(* Logix 5000 project; controller DispersionPlc vendor 1 type 14 code 108 rev 34.11; software revision 34.01; part 14 of 22 *)
(* tags used below, declared in another part *)
   _JISdebug : DINT;
   AFI : BOOL;
   Circulation_Timer_Continue : BOOL;
   Estop_Disp : ALIAS FOR Local:3:I.Data.1;
   FC_4302_1 : AStd_PIDInterface;
   FC_4302_1_AOI : AStd_PIDInterface_AOI;
   FC_4302_1_PID : PID_ENHANCED;
   FC_4305_xx : AStd_PIDInterface;
   FC_4305_xx_AOI : AStd_PIDInterface_AOI;
   FC_4305_xx_PID : PID_ENHANCED;
   FCV_4302_1 : AStd_VlvModulating;
   FIT_4302_2 : AStd_AnalogInput;
   FIT_4305_xx : AStd_AnalogInput;
   FQIC_4302_11_Calc_TransferSetpoint : DINT;
   FQIC_4302_11_CurrentTrasferredLb : DINT;
   FQIC_4302_11_Pulse : BOOL;
   FQIC_4302_11_PulseCounter : COUNTER;
   FQIC_4302_11_PulseToLbFactor : DINT;
   FQIC_4302_11_Reset : BOOL;
   FQIC_4302_11_TransferOffset : DINT;
   FQIC_4302_11_TransferSetpoint : DINT;
   FQIC_4302_11_TransferStopValueLb : DINT;
   FV_4305_xx : AStd_VlvModulating;
   GenPurp : AStd_GeneralPurp;
   LS_4302_High : BOOL;
   One_Shots : DINT;
   P_4305 : AStd_FVNR;
   P_S52_2_OpenC : ALIAS FOR Local:1:O.Data[12].14;
   PLCStatus : AStd_PLCStatus;
   PUMP_P_4305_AUX : ALIAS FOR Local:1:I.Data[1].7;
   RO_END : TIMER;
   RO_HE4305_PhaseROHotWaterDrop : AStd_PLI;
   RO_HE4305_PhaseROWaterAddition : AStd_PLI;
   RO_HE4305_PhaseROWaterAddition_AOI : AStd_PLI_AOI;
   RO_Preheat_Temp : DINT;
   ROWaterAdd_StepComplete : BOOL[32];
   S4352_Phase_Circulation : AStd_PLI;
   S4352_Phase_Circulation_AOI : AStd_PLI_AOI;
   S4352_Phase_Packaging_Transfer : AStd_PLI;
   S4352_Phase_TT_Transfer : AStd_PLI;
   S52_Circulation_StopPB : BOOL;
   S52_Circulation_Timer : TIMER;
   S52CirculationRemMins : REAL;
   SV_4302_1 : AStd_VlvOC;
   SV_4302_1_ICls : BOOL;
   SV_4302_1_IOls : BOOL;
   SV_4302_1_OClose : BOOL;
   SV_S52_2 : AStd_VlvOC;
   SV_S52_2_AOI : AStd_VlvOC_AOI;
   T4302_Phase_S52_Transfer : AStd_PLI;
   T4302_Phase_TT_Transfer : AStd_PLI;
   TC_4305_1 : AStd_PIDInterface;
   TC_4305_1_AOI : AStd_PIDInterface_AOI;
   TC_4305_1_PID : PID_ENHANCED;
   TCV_4305_1 : AStd_VlvModulating;
   TIT_4305_1 : AStd_AnalogInput;
   V4306_PhaseRunPumpCirculate : AStd_PLI;
   V4306_PhaseRunPumpDrumAdd : AStd_PLI;
   V4306_PhaseTransfer : AStd_PLI;
   V4307_PhaseRunPumpCirculate : AStd_PLI;
   V4307_PhaseTransfer : AStd_PLI;
   WIT_4302_1 : AStd_AnalogInput;
   WIT_4306_1 : AStd_AnalogInput;
   WIT_4307_1 : AStd_AnalogInput;
   XV_4301_8 : AStd_VlvOC;
   XV_4302_10 : AStd_VlvOC;
   XV_4302_12 : AStd_VlvOC;
   XV_4302_13 : AStd_VlvOC;
   XV_4302_8 : AStd_VlvOC;
   XV_4306_3 : AStd_VlvOC;
   XV_4306_5 : AStd_VlvOC;
   XV_4307_3 : AStd_VlvOC;
   XV_4307_6 : AStd_VlvOC;
   XV_S52_1 : AStd_VlvOC;
   XV_S52_1_AOI : AStd_VlvOC_AOI;
   XV_S52_1_ClosedI : ALIAS FOR Local:1:I.Data[27].21;
   XV_S52_1_OCls : BOOL;
   XV_S52_1_OpenC : ALIAS FOR Local:1:O.Data[12].16;
   XV_S52_1_OpenI : ALIAS FOR Local:1:I.Data[27].22;
   XV_S52_2 : AStd_VlvOC;
   XV_S52_2_AOI : AStd_VlvOC_AOI;
   XV_S52_2_ClosedI : ALIAS FOR Local:1:I.Data[27].25;
   XV_S52_2_OCls : BOOL;
   XV_S52_2_OpenC : ALIAS FOR Local:1:O.Data[12].18;
   XV_S52_2_OpenI : ALIAS FOR Local:1:I.Data[27].26;
(* Unit_RO_HE4305, continued *)

ROUTINE Phase_ROWaterAddition   (* ladder *)
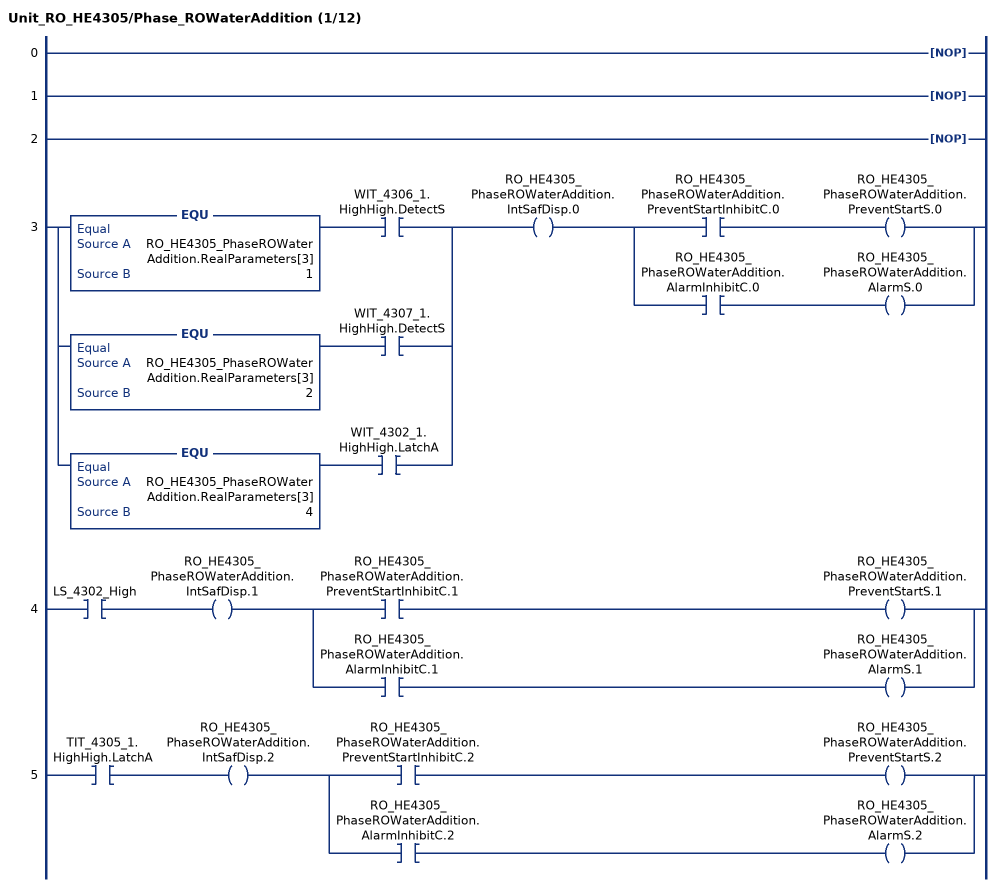
   0: NOP();
   1: NOP();
   2: NOP();
   3: [EQU(RO_HE4305_PhaseROWaterAddition.RealParameters[3],1) XIC(WIT_4306_1.HighHigh.DetectS) ,EQU(RO_HE4305_PhaseROWaterAddition.RealParameters[3],2) XIC(WIT_4307_1.HighHigh.DetectS) ,EQU(RO_HE4305_PhaseROWaterAddition.RealParameters[3],4) XIC(WIT_4302_1.HighHigh.LatchA) ]OTE(RO_HE4305_PhaseROWaterAddition.IntSafDisp.0)[XIC(RO_HE4305_PhaseROWaterAddition.PreventStartInhibitC.0) OTE(RO_HE4305_PhaseROWaterAddition.PreventStartS.0) ,XIC(RO_HE4305_PhaseROWaterAddition.AlarmInhibitC.0) OTE(RO_HE4305_PhaseROWaterAddition.AlarmS.0) ];
   4: XIC(LS_4302_High)OTE(RO_HE4305_PhaseROWaterAddition.IntSafDisp.1)[XIC(RO_HE4305_PhaseROWaterAddition.PreventStartInhibitC.1) OTE(RO_HE4305_PhaseROWaterAddition.PreventStartS.1) ,XIC(RO_HE4305_PhaseROWaterAddition.AlarmInhibitC.1) OTE(RO_HE4305_PhaseROWaterAddition.AlarmS.1) ];
   5: XIC(TIT_4305_1.HighHigh.LatchA)OTE(RO_HE4305_PhaseROWaterAddition.IntSafDisp.2)[XIC(RO_HE4305_PhaseROWaterAddition.PreventStartInhibitC.2) OTE(RO_HE4305_PhaseROWaterAddition.PreventStartS.2) ,XIC(RO_HE4305_PhaseROWaterAddition.AlarmInhibitC.2) OTE(RO_HE4305_PhaseROWaterAddition.AlarmS.2) ];
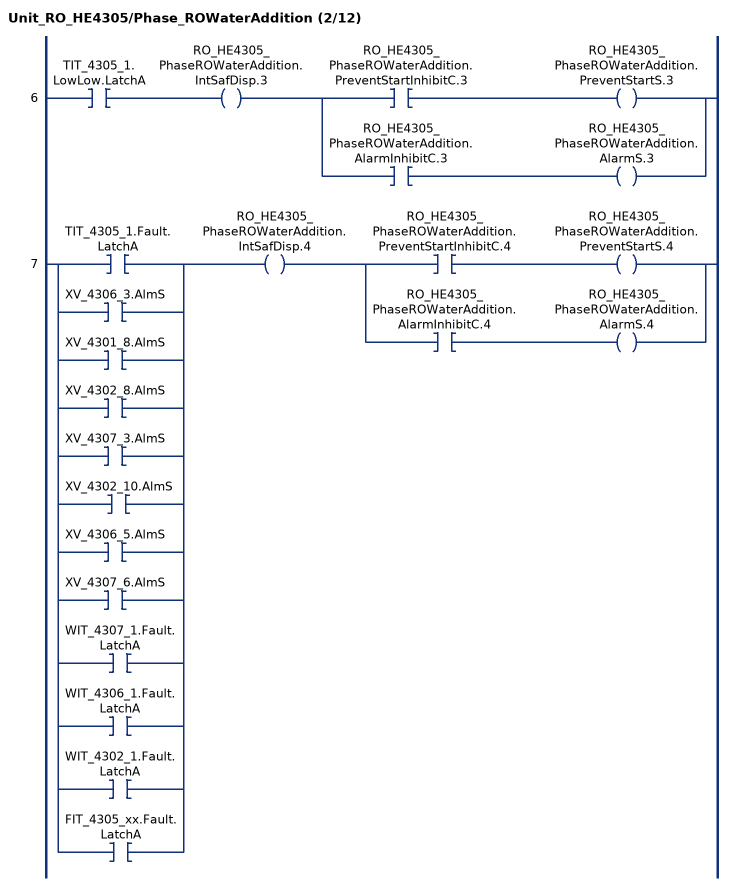
   6: XIC(TIT_4305_1.LowLow.LatchA)OTE(RO_HE4305_PhaseROWaterAddition.IntSafDisp.3)[XIC(RO_HE4305_PhaseROWaterAddition.PreventStartInhibitC.3) OTE(RO_HE4305_PhaseROWaterAddition.PreventStartS.3) ,XIC(RO_HE4305_PhaseROWaterAddition.AlarmInhibitC.3) OTE(RO_HE4305_PhaseROWaterAddition.AlarmS.3) ];
   7: [XIC(TIT_4305_1.Fault.LatchA) ,XIC(XV_4306_3.AlmS) ,XIC(XV_4301_8.AlmS) ,XIC(XV_4302_8.AlmS) ,XIC(XV_4307_3.AlmS) ,XIC(XV_4302_10.AlmS) ,XIC(XV_4306_5.AlmS) ,XIC(XV_4307_6.AlmS) ,XIC(WIT_4307_1.Fault.LatchA) ,XIC(WIT_4306_1.Fault.LatchA) ,XIC(WIT_4302_1.Fault.LatchA) ,XIC(FIT_4305_xx.Fault.LatchA) ]OTE(RO_HE4305_PhaseROWaterAddition.IntSafDisp.4)[XIC(RO_HE4305_PhaseROWaterAddition.PreventStartInhibitC.4) OTE(RO_HE4305_PhaseROWaterAddition.PreventStartS.4) ,XIC(RO_HE4305_PhaseROWaterAddition.AlarmInhibitC.4) OTE(RO_HE4305_PhaseROWaterAddition.AlarmS.4) ];
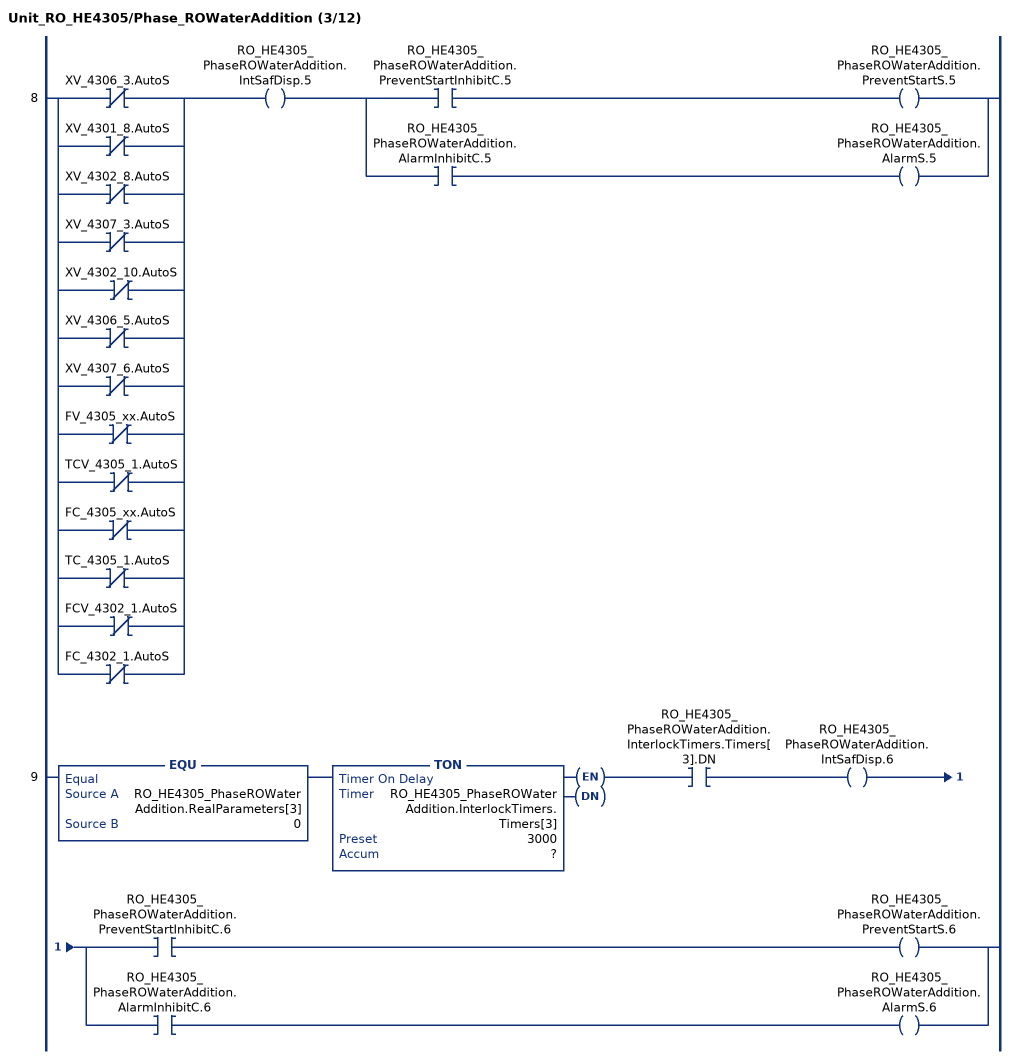
   8: [XIO(XV_4306_3.AutoS) ,XIO(XV_4301_8.AutoS) ,XIO(XV_4302_8.AutoS) ,XIO(XV_4307_3.AutoS) ,XIO(XV_4302_10.AutoS) ,XIO(XV_4306_5.AutoS) ,XIO(XV_4307_6.AutoS) ,XIO(FV_4305_xx.AutoS) ,XIO(TCV_4305_1.AutoS) ,XIO(FC_4305_xx.AutoS) ,XIO(TC_4305_1.AutoS) ,XIO(FCV_4302_1.AutoS) ,XIO(FC_4302_1.AutoS) ]OTE(RO_HE4305_PhaseROWaterAddition.IntSafDisp.5)[XIC(RO_HE4305_PhaseROWaterAddition.PreventStartInhibitC.5) OTE(RO_HE4305_PhaseROWaterAddition.PreventStartS.5) ,XIC(RO_HE4305_PhaseROWaterAddition.AlarmInhibitC.5) OTE(RO_HE4305_PhaseROWaterAddition.AlarmS.5) ];
   9: EQU(RO_HE4305_PhaseROWaterAddition.RealParameters[3],0)TON(RO_HE4305_PhaseROWaterAddition.InterlockTimers.Timers[3],?,?)XIC(RO_HE4305_PhaseROWaterAddition.InterlockTimers.Timers[3].DN)OTE(RO_HE4305_PhaseROWaterAddition.IntSafDisp.6)[XIC(RO_HE4305_PhaseROWaterAddition.PreventStartInhibitC.6) OTE(RO_HE4305_PhaseROWaterAddition.PreventStartS.6) ,XIC(RO_HE4305_PhaseROWaterAddition.AlarmInhibitC.6) OTE(RO_HE4305_PhaseROWaterAddition.AlarmS.6) ];
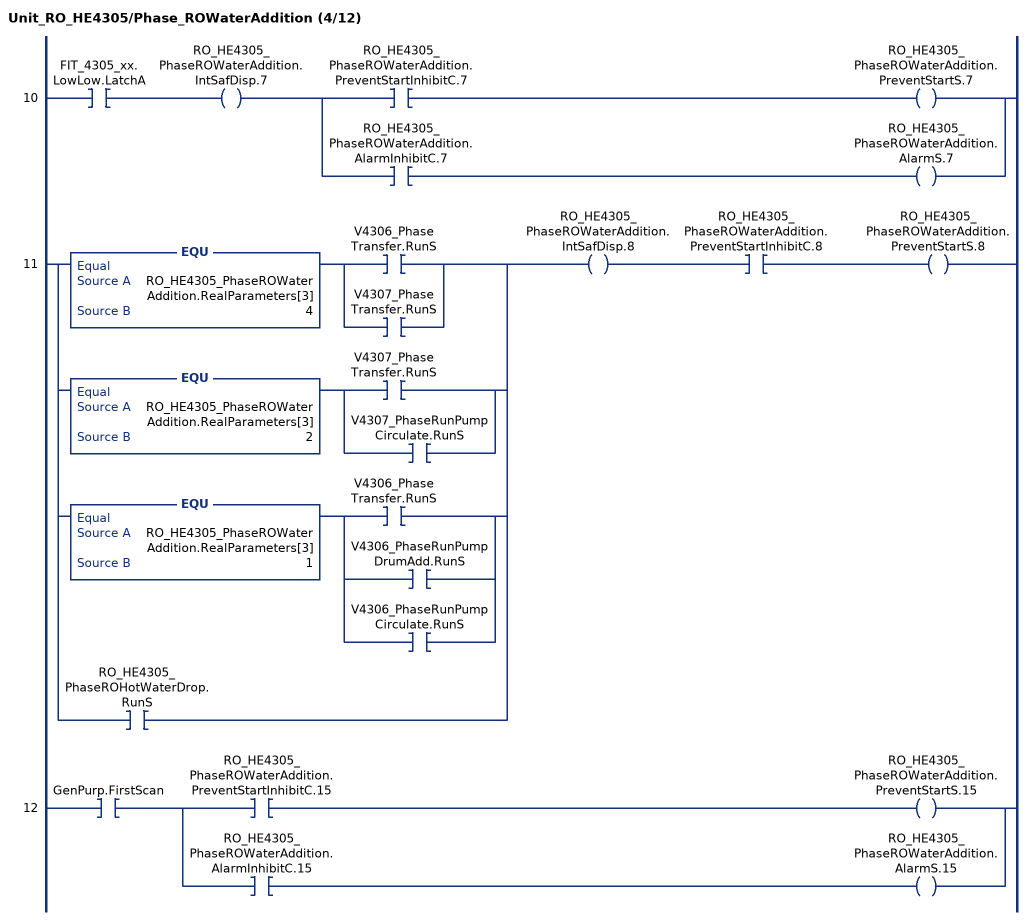
   10: XIC(FIT_4305_xx.LowLow.LatchA)OTE(RO_HE4305_PhaseROWaterAddition.IntSafDisp.7)[XIC(RO_HE4305_PhaseROWaterAddition.PreventStartInhibitC.7) OTE(RO_HE4305_PhaseROWaterAddition.PreventStartS.7) ,XIC(RO_HE4305_PhaseROWaterAddition.AlarmInhibitC.7) OTE(RO_HE4305_PhaseROWaterAddition.AlarmS.7) ];
   11: [EQU(RO_HE4305_PhaseROWaterAddition.RealParameters[3],4) [XIC(V4306_PhaseTransfer.RunS) ,XIC(V4307_PhaseTransfer.RunS) ] ,EQU(RO_HE4305_PhaseROWaterAddition.RealParameters[3],2) [XIC(V4307_PhaseTransfer.RunS) ,XIC(V4307_PhaseRunPumpCirculate.RunS) ] ,EQU(RO_HE4305_PhaseROWaterAddition.RealParameters[3],1) [XIC(V4306_PhaseTransfer.RunS) ,XIC(V4306_PhaseRunPumpDrumAdd.RunS) ,XIC(V4306_PhaseRunPumpCirculate.RunS) ] ,XIC(RO_HE4305_PhaseROHotWaterDrop.RunS) ]OTE(RO_HE4305_PhaseROWaterAddition.IntSafDisp.8)XIC(RO_HE4305_PhaseROWaterAddition.PreventStartInhibitC.8)OTE(RO_HE4305_PhaseROWaterAddition.PreventStartS.8);
   12: XIC(GenPurp.FirstScan)[XIC(RO_HE4305_PhaseROWaterAddition.PreventStartInhibitC.15) OTE(RO_HE4305_PhaseROWaterAddition.PreventStartS.15) ,XIC(RO_HE4305_PhaseROWaterAddition.AlarmInhibitC.15) OTE(RO_HE4305_PhaseROWaterAddition.AlarmS.15) ];
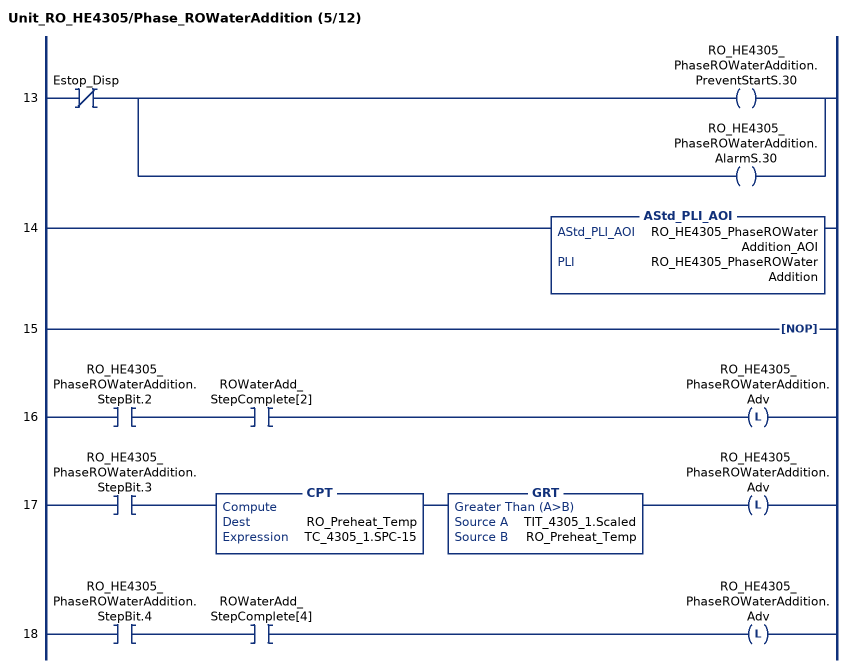
   13: XIO(Estop_Disp)[OTE(RO_HE4305_PhaseROWaterAddition.PreventStartS.30) ,OTE(RO_HE4305_PhaseROWaterAddition.AlarmS.30) ];
   14: AStd_PLI_AOI(RO_HE4305_PhaseROWaterAddition_AOI,RO_HE4305_PhaseROWaterAddition);
   15: NOP();
   16: XIC(RO_HE4305_PhaseROWaterAddition.StepBit.2)XIC(ROWaterAdd_StepComplete[2])OTL(RO_HE4305_PhaseROWaterAddition.Adv);
   17: XIC(RO_HE4305_PhaseROWaterAddition.StepBit.3)CPT(RO_Preheat_Temp,TC_4305_1.SPC-15)GRT(TIT_4305_1.Scaled,RO_Preheat_Temp)OTL(RO_HE4305_PhaseROWaterAddition.Adv);
   18: XIC(RO_HE4305_PhaseROWaterAddition.StepBit.4)XIC(ROWaterAdd_StepComplete[4])OTL(RO_HE4305_PhaseROWaterAddition.Adv);
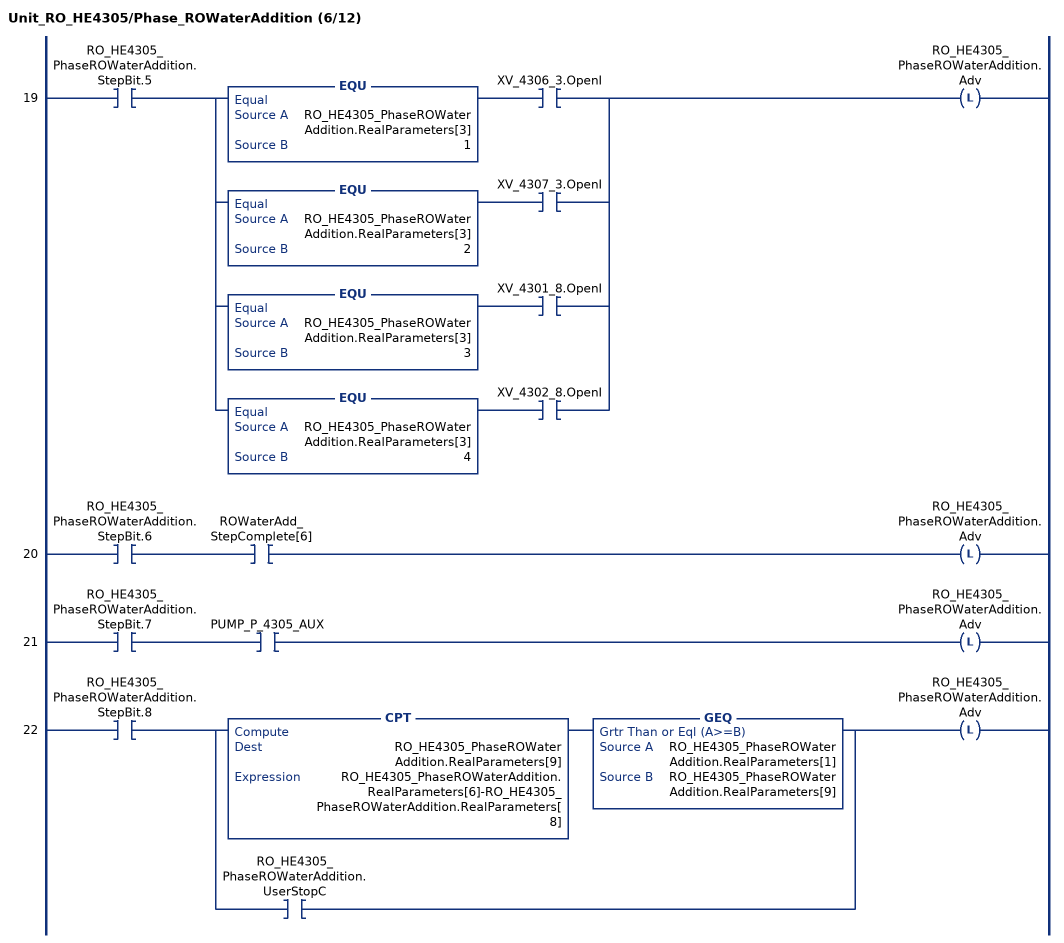
   19: XIC(RO_HE4305_PhaseROWaterAddition.StepBit.5)[EQU(RO_HE4305_PhaseROWaterAddition.RealParameters[3],1) XIC(XV_4306_3.OpenI) ,EQU(RO_HE4305_PhaseROWaterAddition.RealParameters[3],2) XIC(XV_4307_3.OpenI) ,EQU(RO_HE4305_PhaseROWaterAddition.RealParameters[3],3) XIC(XV_4301_8.OpenI) ,EQU(RO_HE4305_PhaseROWaterAddition.RealParameters[3],4) XIC(XV_4302_8.OpenI) ]OTL(RO_HE4305_PhaseROWaterAddition.Adv);
   20: XIC(RO_HE4305_PhaseROWaterAddition.StepBit.6)XIC(ROWaterAdd_StepComplete[6])OTL(RO_HE4305_PhaseROWaterAddition.Adv);
   21: XIC(RO_HE4305_PhaseROWaterAddition.StepBit.7)XIC(PUMP_P_4305_AUX)OTL(RO_HE4305_PhaseROWaterAddition.Adv);
   22: XIC(RO_HE4305_PhaseROWaterAddition.StepBit.8)[CPT(RO_HE4305_PhaseROWaterAddition.RealParameters[9],RO_HE4305_PhaseROWaterAddition.RealParameters[6]-RO_HE4305_PhaseROWaterAddition.RealParameters[8]) GEQ(RO_HE4305_PhaseROWaterAddition.RealParameters[1],RO_HE4305_PhaseROWaterAddition.RealParameters[9]) ,XIC(RO_HE4305_PhaseROWaterAddition.UserStopC) ]OTL(RO_HE4305_PhaseROWaterAddition.Adv);
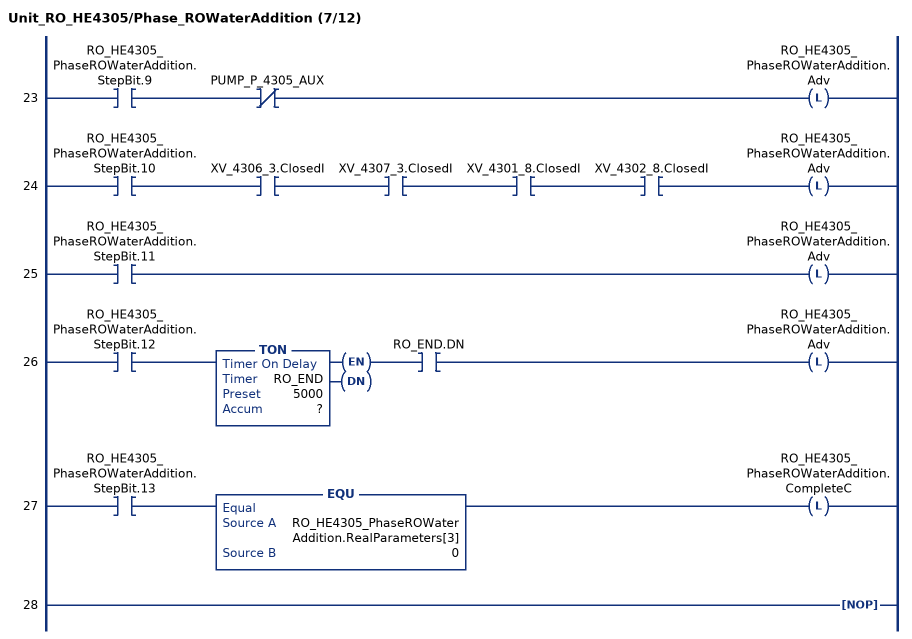
   23: XIC(RO_HE4305_PhaseROWaterAddition.StepBit.9)XIO(PUMP_P_4305_AUX)OTL(RO_HE4305_PhaseROWaterAddition.Adv);
   24: XIC(RO_HE4305_PhaseROWaterAddition.StepBit.10)XIC(XV_4306_3.ClosedI)XIC(XV_4307_3.ClosedI)XIC(XV_4301_8.ClosedI)XIC(XV_4302_8.ClosedI)OTL(RO_HE4305_PhaseROWaterAddition.Adv);
   25: XIC(RO_HE4305_PhaseROWaterAddition.StepBit.11)OTL(RO_HE4305_PhaseROWaterAddition.Adv);
   26: XIC(RO_HE4305_PhaseROWaterAddition.StepBit.12)TON(RO_END,?,?)XIC(RO_END.DN)OTL(RO_HE4305_PhaseROWaterAddition.Adv);
   27: XIC(RO_HE4305_PhaseROWaterAddition.StepBit.13)EQU(RO_HE4305_PhaseROWaterAddition.RealParameters[3],0)OTL(RO_HE4305_PhaseROWaterAddition.CompleteC);
   28: NOP();
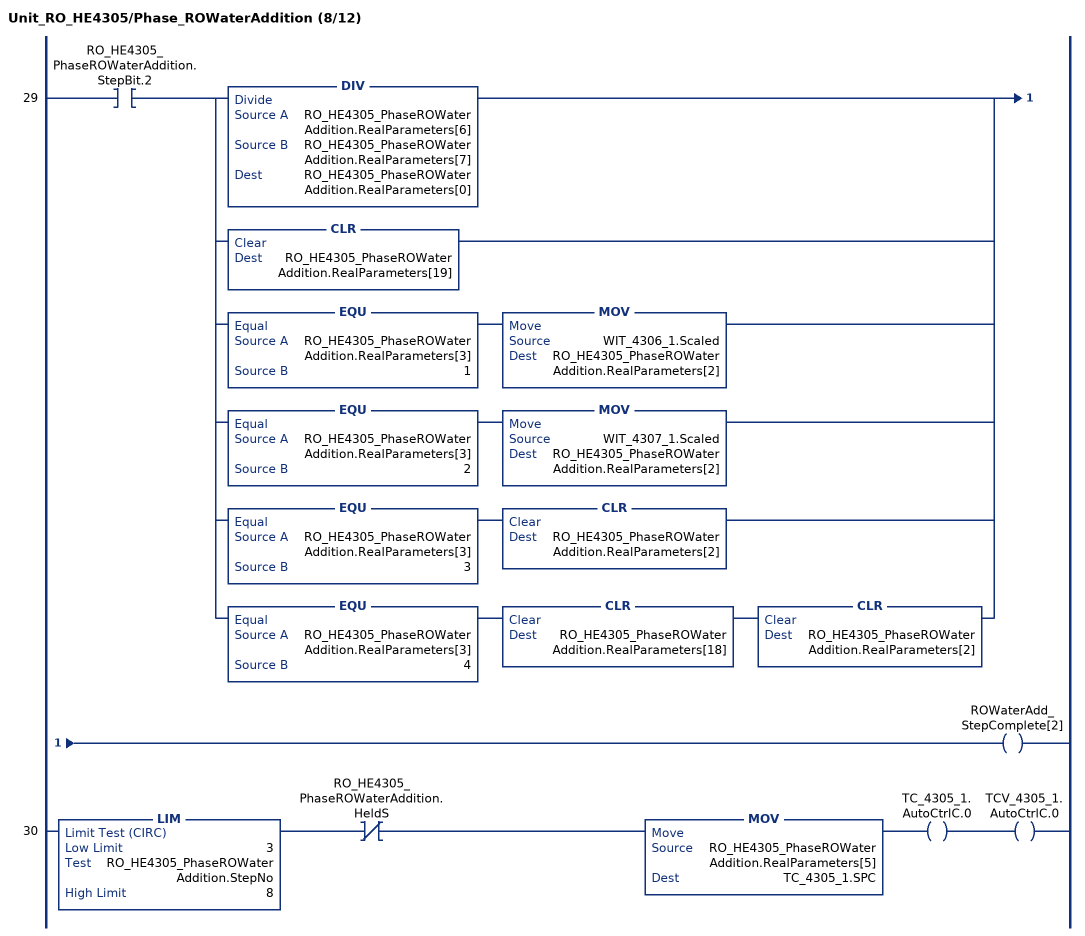
   29: XIC(RO_HE4305_PhaseROWaterAddition.StepBit.2)[DIV(RO_HE4305_PhaseROWaterAddition.RealParameters[6],RO_HE4305_PhaseROWaterAddition.RealParameters[7],RO_HE4305_PhaseROWaterAddition.RealParameters[0]) ,CLR(RO_HE4305_PhaseROWaterAddition.RealParameters[19]) ,EQU(RO_HE4305_PhaseROWaterAddition.RealParameters[3],1) MOV(WIT_4306_1.Scaled,RO_HE4305_PhaseROWaterAddition.RealParameters[2]) ,EQU(RO_HE4305_PhaseROWaterAddition.RealParameters[3],2) MOV(WIT_4307_1.Scaled,RO_HE4305_PhaseROWaterAddition.RealParameters[2]) ,EQU(RO_HE4305_PhaseROWaterAddition.RealParameters[3],3) CLR(RO_HE4305_PhaseROWaterAddition.RealParameters[2]) ,EQU(RO_HE4305_PhaseROWaterAddition.RealParameters[3],4) CLR(RO_HE4305_PhaseROWaterAddition.RealParameters[18]) CLR(RO_HE4305_PhaseROWaterAddition.RealParameters[2]) ]OTE(ROWaterAdd_StepComplete[2]);
   30: LIM(3,RO_HE4305_PhaseROWaterAddition.StepNo,8)XIO(RO_HE4305_PhaseROWaterAddition.HeldS)MOV(RO_HE4305_PhaseROWaterAddition.RealParameters[5],TC_4305_1.SPC)OTE(TC_4305_1.AutoCtrlC.0)OTE(TCV_4305_1.AutoCtrlC.0);
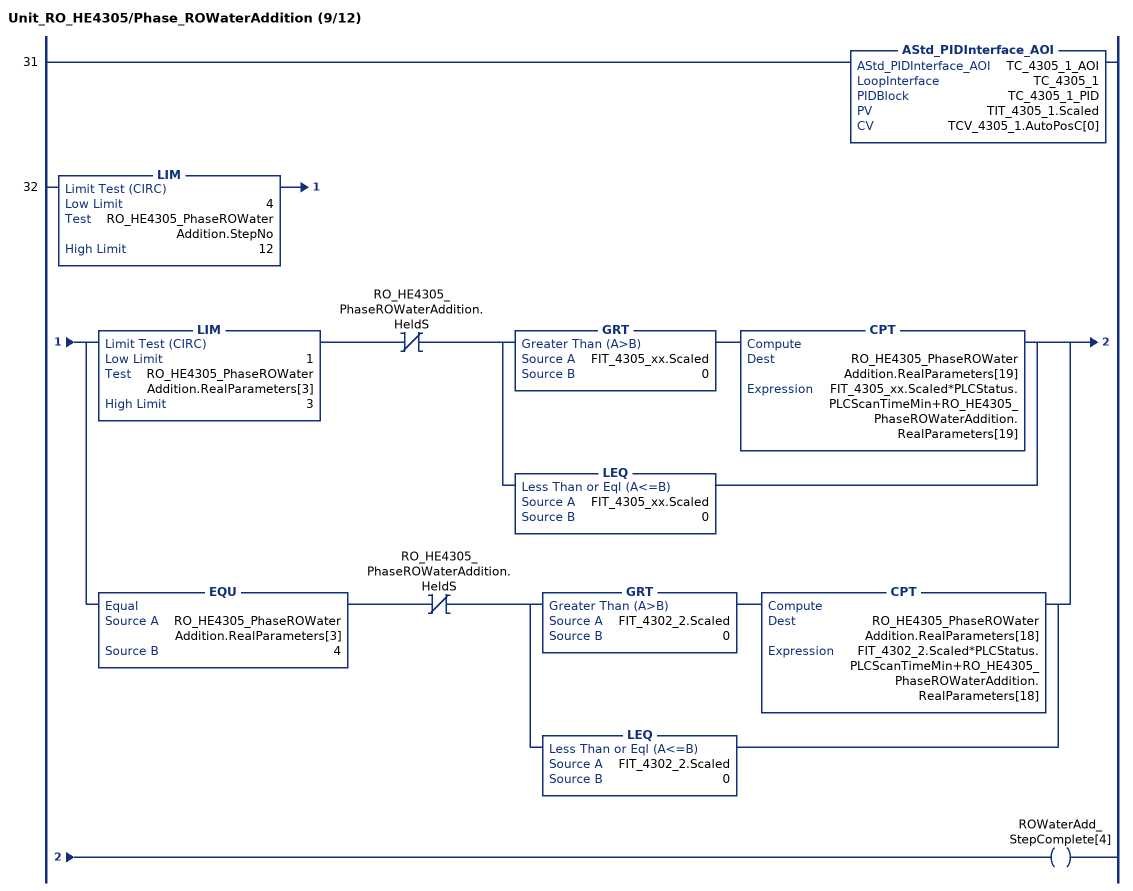
   31: AStd_PIDInterface_AOI(TC_4305_1_AOI,TC_4305_1,TC_4305_1_PID,TIT_4305_1.Scaled,TCV_4305_1.AutoPosC[0]);
   32: LIM(4,RO_HE4305_PhaseROWaterAddition.StepNo,12)[LIM(1,RO_HE4305_PhaseROWaterAddition.RealParameters[3],3) XIO(RO_HE4305_PhaseROWaterAddition.HeldS) [GRT(FIT_4305_xx.Scaled,0) CPT(RO_HE4305_PhaseROWaterAddition.RealParameters[19],FIT_4305_xx.Scaled*PLCStatus.PLCScanTimeMin+RO_HE4305_PhaseROWaterAddition.RealParameters[19]) ,LEQ(FIT_4305_xx.Scaled,0) ] ,EQU(RO_HE4305_PhaseROWaterAddition.RealParameters[3],4) XIO(RO_HE4305_PhaseROWaterAddition.HeldS) [GRT(FIT_4302_2.Scaled,0) CPT(RO_HE4305_PhaseROWaterAddition.RealParameters[18],FIT_4302_2.Scaled*PLCStatus.PLCScanTimeMin+RO_HE4305_PhaseROWaterAddition.RealParameters[18]) ,LEQ(FIT_4302_2.Scaled,0) ] ]OTE(ROWaterAdd_StepComplete[4]);
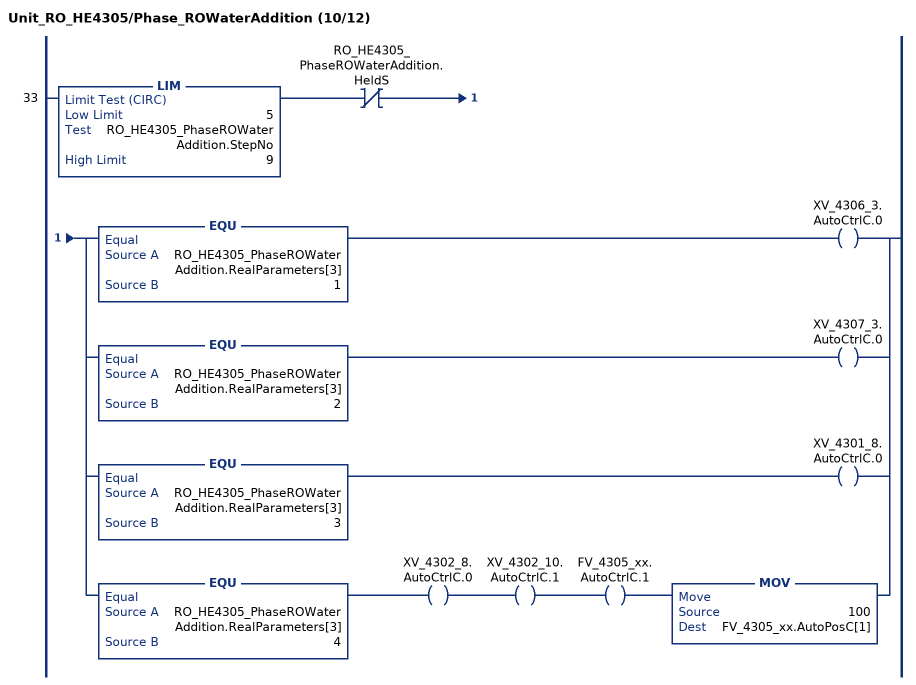
   33: LIM(5,RO_HE4305_PhaseROWaterAddition.StepNo,9)XIO(RO_HE4305_PhaseROWaterAddition.HeldS)[EQU(RO_HE4305_PhaseROWaterAddition.RealParameters[3],1) OTE(XV_4306_3.AutoCtrlC.0) ,EQU(RO_HE4305_PhaseROWaterAddition.RealParameters[3],2) OTE(XV_4307_3.AutoCtrlC.0) ,EQU(RO_HE4305_PhaseROWaterAddition.RealParameters[3],3) OTE(XV_4301_8.AutoCtrlC.0) ,EQU(RO_HE4305_PhaseROWaterAddition.RealParameters[3],4) OTE(XV_4302_8.AutoCtrlC.0) OTE(XV_4302_10.AutoCtrlC.1) OTE(FV_4305_xx.AutoCtrlC.1) MOV(100,FV_4305_xx.AutoPosC[1]) ];
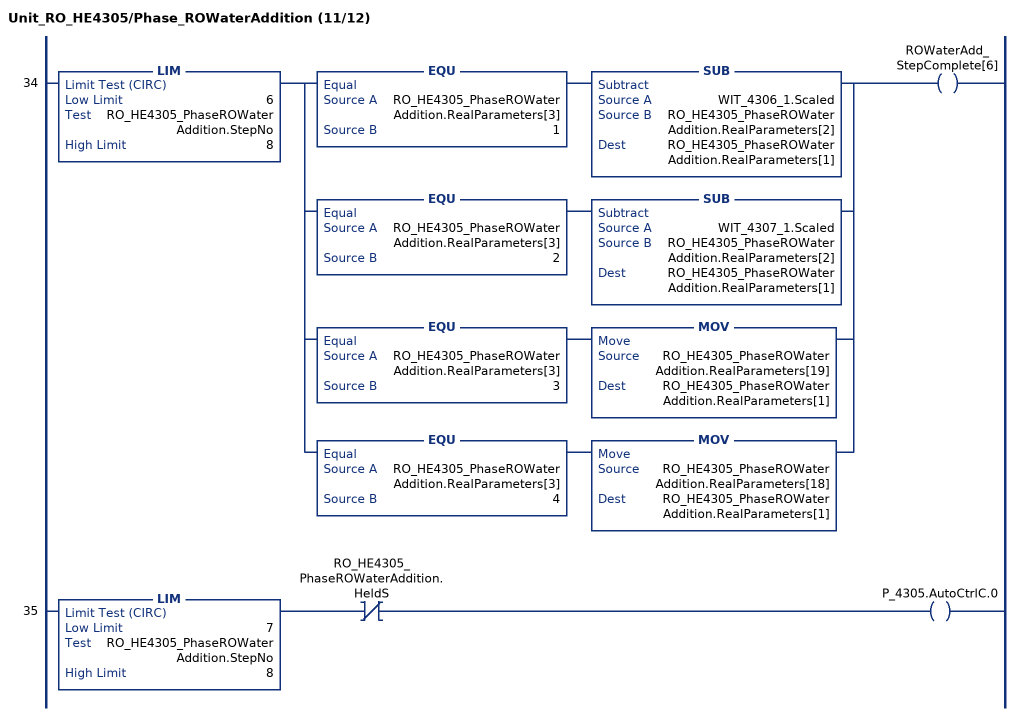
   34: LIM(6,RO_HE4305_PhaseROWaterAddition.StepNo,8)[EQU(RO_HE4305_PhaseROWaterAddition.RealParameters[3],1) SUB(WIT_4306_1.Scaled,RO_HE4305_PhaseROWaterAddition.RealParameters[2],RO_HE4305_PhaseROWaterAddition.RealParameters[1]) ,EQU(RO_HE4305_PhaseROWaterAddition.RealParameters[3],2) SUB(WIT_4307_1.Scaled,RO_HE4305_PhaseROWaterAddition.RealParameters[2],RO_HE4305_PhaseROWaterAddition.RealParameters[1]) ,EQU(RO_HE4305_PhaseROWaterAddition.RealParameters[3],3) MOV(RO_HE4305_PhaseROWaterAddition.RealParameters[19],RO_HE4305_PhaseROWaterAddition.RealParameters[1]) ,EQU(RO_HE4305_PhaseROWaterAddition.RealParameters[3],4) MOV(RO_HE4305_PhaseROWaterAddition.RealParameters[18],RO_HE4305_PhaseROWaterAddition.RealParameters[1]) ]OTE(ROWaterAdd_StepComplete[6]);
   35: LIM(7,RO_HE4305_PhaseROWaterAddition.StepNo,8)XIO(RO_HE4305_PhaseROWaterAddition.HeldS)OTE(P_4305.AutoCtrlC.0);
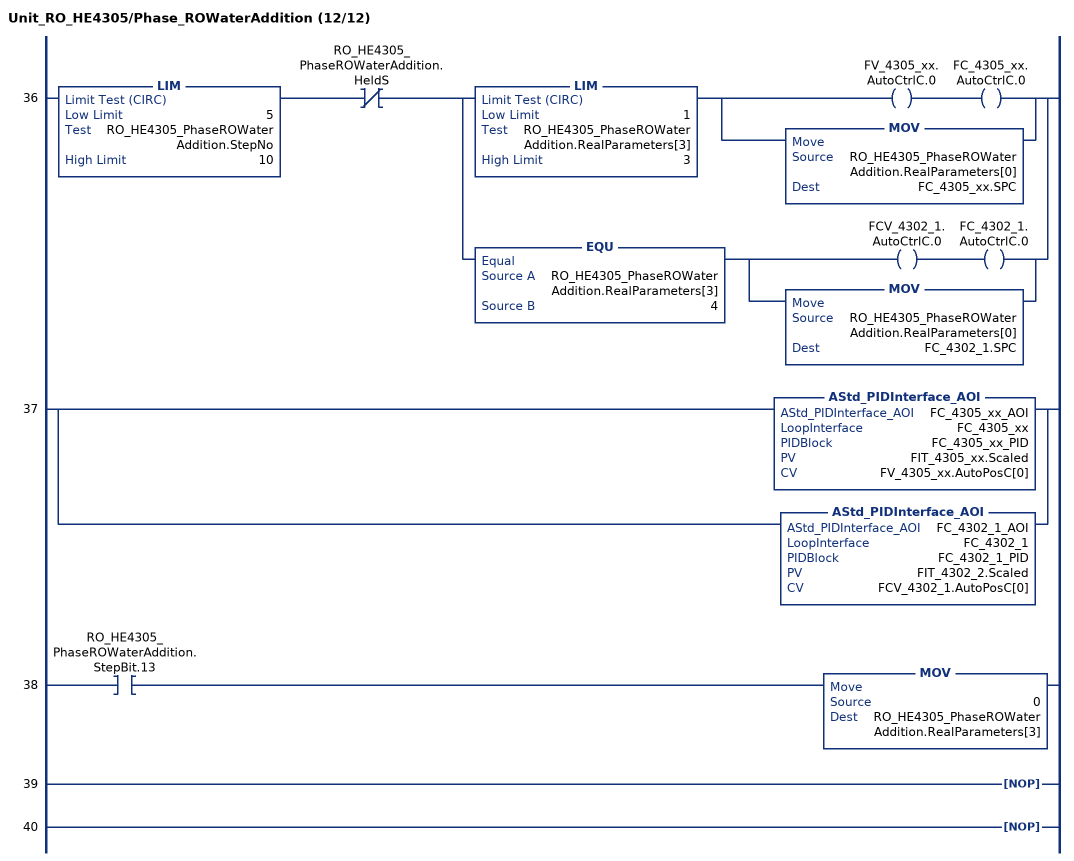
   36: LIM(5,RO_HE4305_PhaseROWaterAddition.StepNo,10)XIO(RO_HE4305_PhaseROWaterAddition.HeldS)[LIM(1,RO_HE4305_PhaseROWaterAddition.RealParameters[3],3) [OTE(FV_4305_xx.AutoCtrlC.0) OTE(FC_4305_xx.AutoCtrlC.0) ,MOV(RO_HE4305_PhaseROWaterAddition.RealParameters[0],FC_4305_xx.SPC) ] ,EQU(RO_HE4305_PhaseROWaterAddition.RealParameters[3],4) [OTE(FCV_4302_1.AutoCtrlC.0) OTE(FC_4302_1.AutoCtrlC.0) ,MOV(RO_HE4305_PhaseROWaterAddition.RealParameters[0],FC_4302_1.SPC) ] ];
   37: [AStd_PIDInterface_AOI(FC_4305_xx_AOI,FC_4305_xx,FC_4305_xx_PID,FIT_4305_xx.Scaled,FV_4305_xx.AutoPosC[0]) ,AStd_PIDInterface_AOI(FC_4302_1_AOI,FC_4302_1,FC_4302_1_PID,FIT_4302_2.Scaled,FCV_4302_1.AutoPosC[0]) ];
   38: XIC(RO_HE4305_PhaseROWaterAddition.StepBit.13)MOV(0,RO_HE4305_PhaseROWaterAddition.RealParameters[3]);
   39: NOP();
   40: NOP();
END_ROUTINE
END_PROGRAM

PROGRAM Unit_S4352   (* main routine MainRoutine *)

ROUTINE Device_SV_S52_2   (* ladder *)
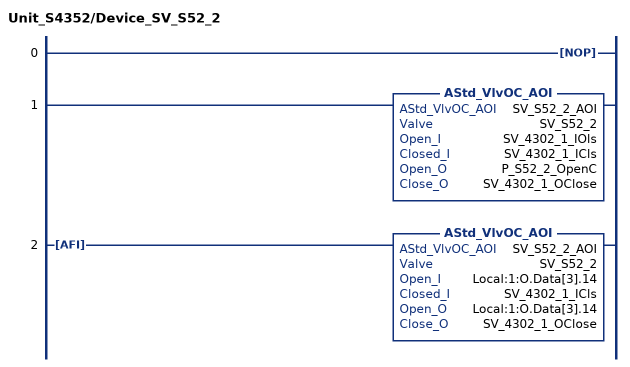
   0: NOP();
   1: AStd_VlvOC_AOI(SV_S52_2_AOI,SV_S52_2,SV_4302_1_IOls,SV_4302_1_ICls,P_S52_2_OpenC,SV_4302_1_OClose);
   2: AFI()AStd_VlvOC_AOI(SV_S52_2_AOI,SV_S52_2,Local:1:O.Data[3].14,SV_4302_1_ICls,Local:1:O.Data[3].14,SV_4302_1_OClose);
END_ROUTINE

ROUTINE Device_XV_S52_1   (* ladder *)
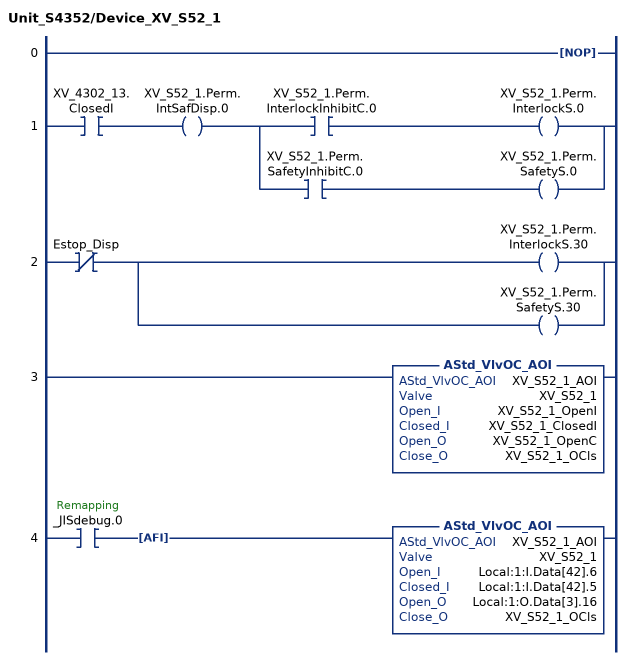
   0: NOP();
   1: XIC(XV_4302_13.ClosedI)OTE(XV_S52_1.Perm.IntSafDisp.0)[XIC(XV_S52_1.Perm.InterlockInhibitC.0) OTE(XV_S52_1.Perm.InterlockS.0) ,XIC(XV_S52_1.Perm.SafetyInhibitC.0) OTE(XV_S52_1.Perm.SafetyS.0) ];
   2: XIO(Estop_Disp)[OTE(XV_S52_1.Perm.InterlockS.30) ,OTE(XV_S52_1.Perm.SafetyS.30) ];
   3: AStd_VlvOC_AOI(XV_S52_1_AOI,XV_S52_1,XV_S52_1_OpenI,XV_S52_1_ClosedI,XV_S52_1_OpenC,XV_S52_1_OCls);
   4: XIC(_JISdebug.0)AFI()AStd_VlvOC_AOI(XV_S52_1_AOI,XV_S52_1,Local:1:I.Data[42].6,Local:1:I.Data[42].5,Local:1:O.Data[3].16,XV_S52_1_OCls);
END_ROUTINE

ROUTINE Device_XV_S52_2   (* ladder *)
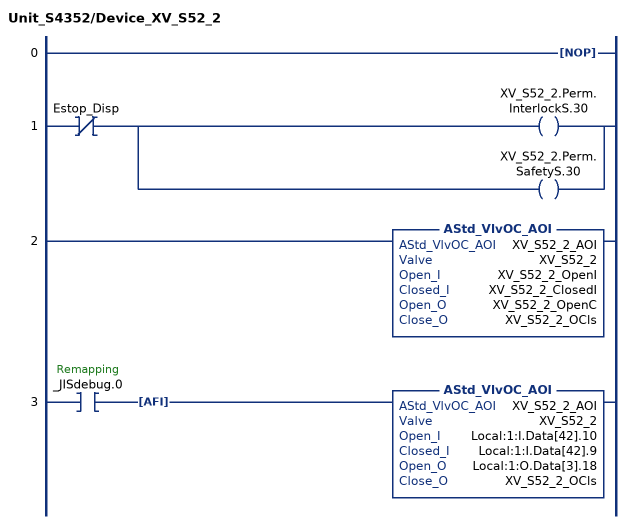
   0: NOP();
   1: XIO(Estop_Disp)[OTE(XV_S52_2.Perm.InterlockS.30) ,OTE(XV_S52_2.Perm.SafetyS.30) ];
   2: AStd_VlvOC_AOI(XV_S52_2_AOI,XV_S52_2,XV_S52_2_OpenI,XV_S52_2_ClosedI,XV_S52_2_OpenC,XV_S52_2_OCls);
   3: XIC(_JISdebug.0)AFI()AStd_VlvOC_AOI(XV_S52_2_AOI,XV_S52_2,Local:1:I.Data[42].10,Local:1:I.Data[42].9,Local:1:O.Data[3].18,XV_S52_2_OCls);
END_ROUTINE

ROUTINE MainRoutine   (* ladder *)
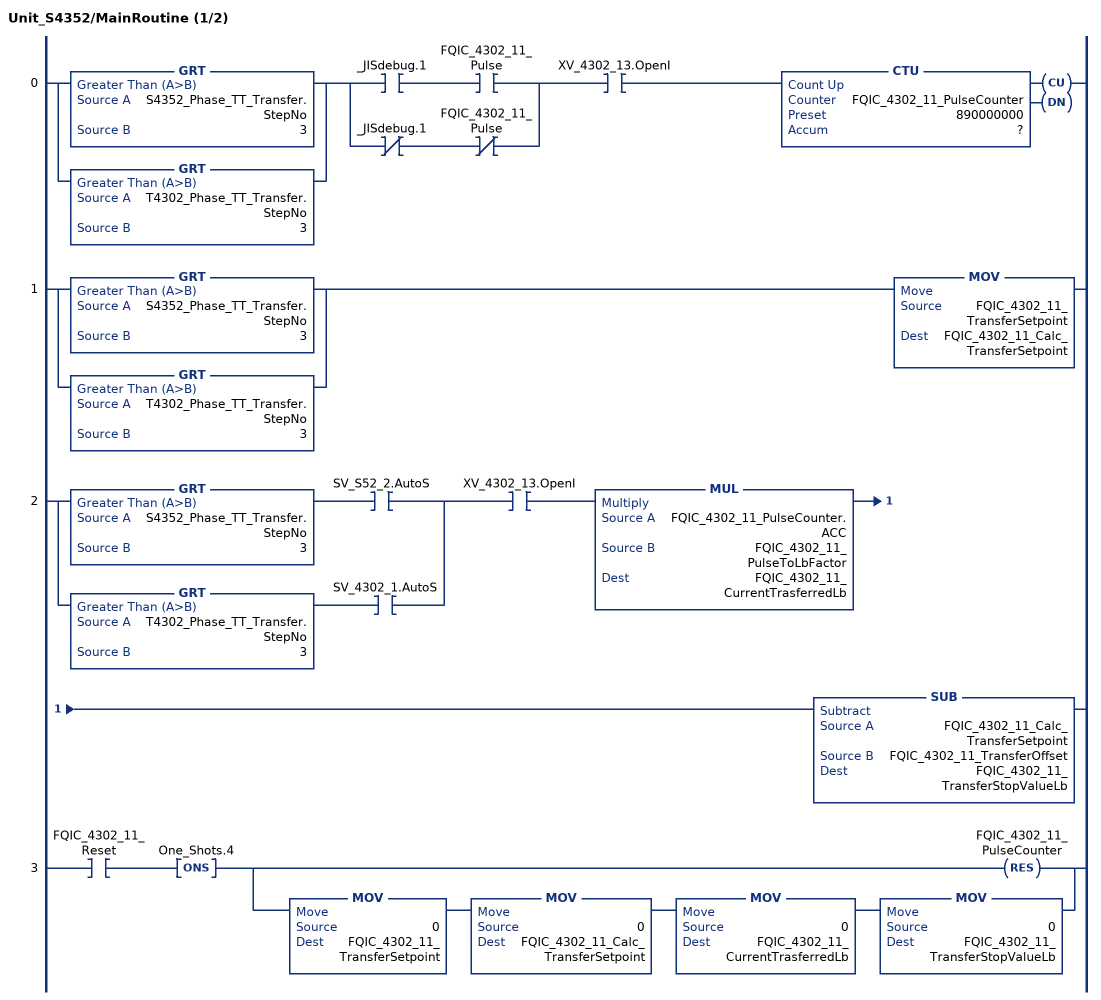
   0: [GRT(S4352_Phase_TT_Transfer.StepNo,3) ,GRT(T4302_Phase_TT_Transfer.StepNo,3) ][XIC(_JISdebug.1) XIC(FQIC_4302_11_Pulse) ,XIO(_JISdebug.1) XIO(FQIC_4302_11_Pulse) ]XIC(XV_4302_13.OpenI)CTU(FQIC_4302_11_PulseCounter,?,?);
   1: [GRT(S4352_Phase_TT_Transfer.StepNo,3) ,GRT(T4302_Phase_TT_Transfer.StepNo,3) ]MOV(FQIC_4302_11_TransferSetpoint,FQIC_4302_11_Calc_TransferSetpoint);
   2: [GRT(S4352_Phase_TT_Transfer.StepNo,3) XIC(SV_S52_2.AutoS) ,GRT(T4302_Phase_TT_Transfer.StepNo,3) XIC(SV_4302_1.AutoS) ]XIC(XV_4302_13.OpenI)MUL(FQIC_4302_11_PulseCounter.ACC,FQIC_4302_11_PulseToLbFactor,FQIC_4302_11_CurrentTrasferredLb)SUB(FQIC_4302_11_Calc_TransferSetpoint,FQIC_4302_11_TransferOffset,FQIC_4302_11_TransferStopValueLb);
   3: XIC(FQIC_4302_11_Reset)ONS(One_Shots.4)[RES(FQIC_4302_11_PulseCounter) ,MOV(0,FQIC_4302_11_TransferSetpoint) MOV(0,FQIC_4302_11_Calc_TransferSetpoint) MOV(0,FQIC_4302_11_CurrentTrasferredLb) MOV(0,FQIC_4302_11_TransferStopValueLb) ];
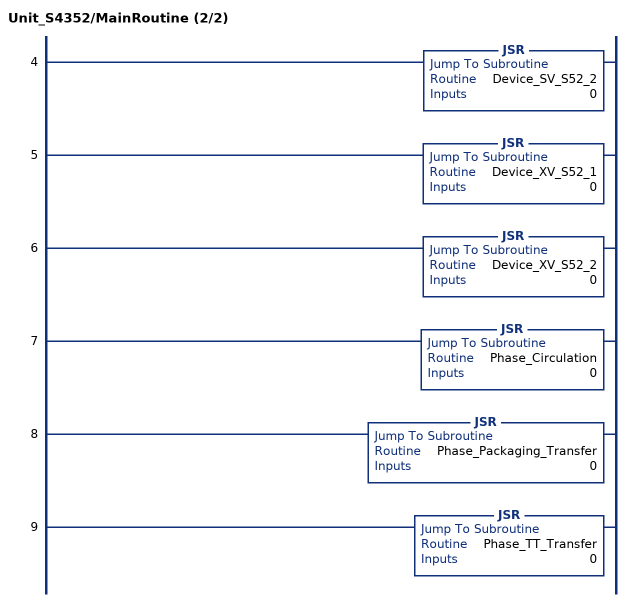
   4: JSR(Device_SV_S52_2,0);
   5: JSR(Device_XV_S52_1,0);
   6: JSR(Device_XV_S52_2,0);
   7: JSR(Phase_Circulation,0);
   8: JSR(Phase_Packaging_Transfer,0);
   9: JSR(Phase_TT_Transfer,0);
END_ROUTINE

ROUTINE Phase_Circulation   (* ladder *)
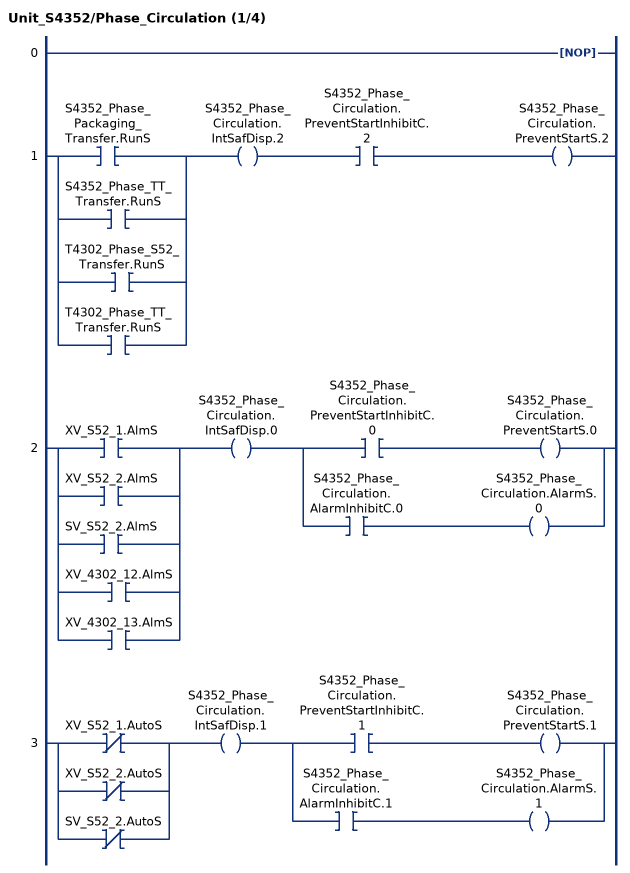
   0: NOP();
   1: [XIC(S4352_Phase_Packaging_Transfer.RunS) ,XIC(S4352_Phase_TT_Transfer.RunS) ,XIC(T4302_Phase_S52_Transfer.RunS) ,XIC(T4302_Phase_TT_Transfer.RunS) ]OTE(S4352_Phase_Circulation.IntSafDisp.2)XIC(S4352_Phase_Circulation.PreventStartInhibitC.2)OTE(S4352_Phase_Circulation.PreventStartS.2);
   2: [XIC(XV_S52_1.AlmS) ,XIC(XV_S52_2.AlmS) ,XIC(SV_S52_2.AlmS) ,XIC(XV_4302_12.AlmS) ,XIC(XV_4302_13.AlmS) ]OTE(S4352_Phase_Circulation.IntSafDisp.0)[XIC(S4352_Phase_Circulation.PreventStartInhibitC.0) OTE(S4352_Phase_Circulation.PreventStartS.0) ,XIC(S4352_Phase_Circulation.AlarmInhibitC.0) OTE(S4352_Phase_Circulation.AlarmS.0) ];
   3: [XIO(XV_S52_1.AutoS) ,XIO(XV_S52_2.AutoS) ,XIO(SV_S52_2.AutoS) ]OTE(S4352_Phase_Circulation.IntSafDisp.1)[XIC(S4352_Phase_Circulation.PreventStartInhibitC.1) OTE(S4352_Phase_Circulation.PreventStartS.1) ,XIC(S4352_Phase_Circulation.AlarmInhibitC.1) OTE(S4352_Phase_Circulation.AlarmS.1) ];
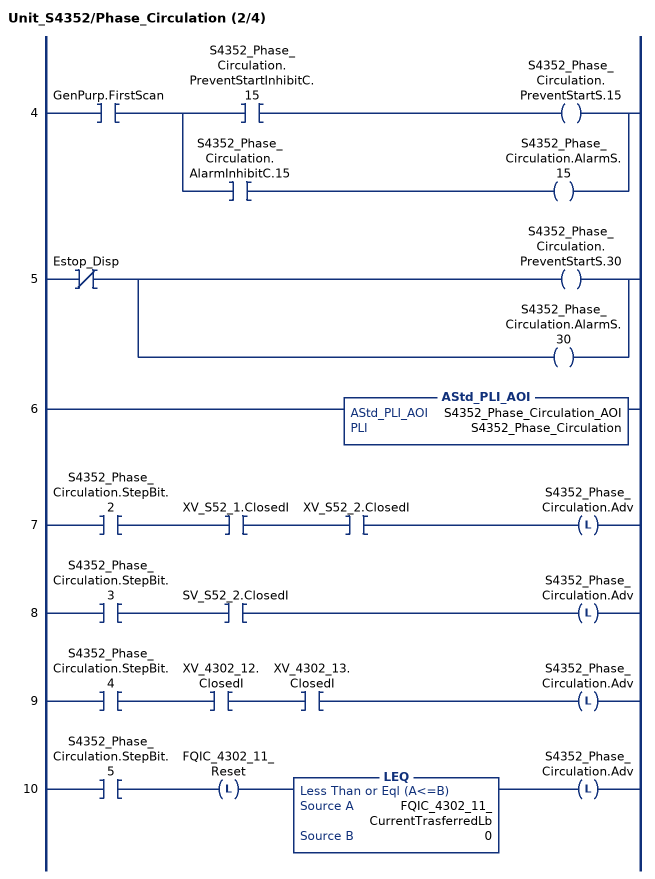
   4: XIC(GenPurp.FirstScan)[XIC(S4352_Phase_Circulation.PreventStartInhibitC.15) OTE(S4352_Phase_Circulation.PreventStartS.15) ,XIC(S4352_Phase_Circulation.AlarmInhibitC.15) OTE(S4352_Phase_Circulation.AlarmS.15) ];
   5: XIO(Estop_Disp)[OTE(S4352_Phase_Circulation.PreventStartS.30) ,OTE(S4352_Phase_Circulation.AlarmS.30) ];
   6: AStd_PLI_AOI(S4352_Phase_Circulation_AOI,S4352_Phase_Circulation);
   7: XIC(S4352_Phase_Circulation.StepBit.2)XIC(XV_S52_1.ClosedI)XIC(XV_S52_2.ClosedI)OTL(S4352_Phase_Circulation.Adv);
   8: XIC(S4352_Phase_Circulation.StepBit.3)XIC(SV_S52_2.ClosedI)OTL(S4352_Phase_Circulation.Adv);
   9: XIC(S4352_Phase_Circulation.StepBit.4)XIC(XV_4302_12.ClosedI)XIC(XV_4302_13.ClosedI)OTL(S4352_Phase_Circulation.Adv);
   10: XIC(S4352_Phase_Circulation.StepBit.5)OTL(FQIC_4302_11_Reset)LEQ(FQIC_4302_11_CurrentTrasferredLb,0)OTL(S4352_Phase_Circulation.Adv);
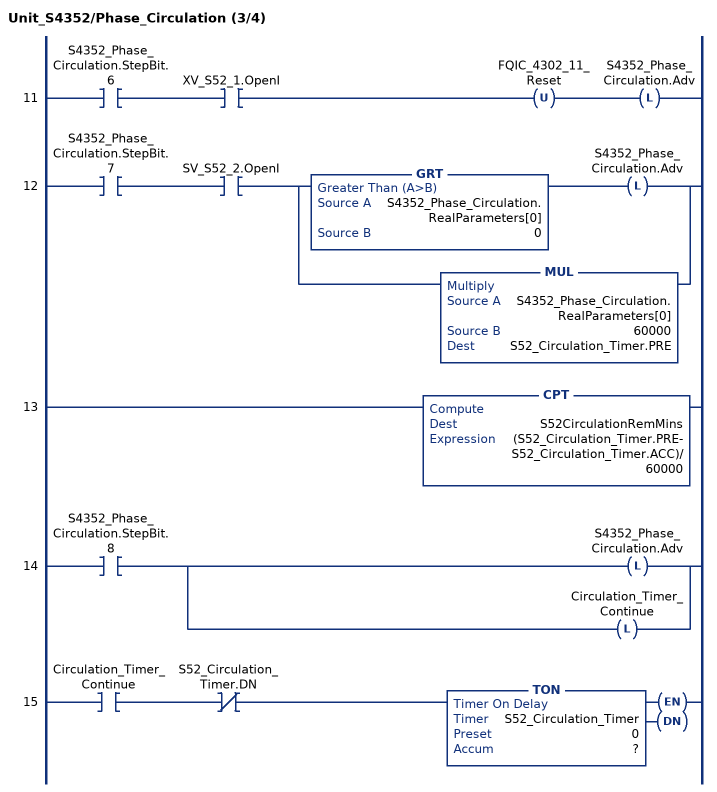
   11: XIC(S4352_Phase_Circulation.StepBit.6)XIC(XV_S52_1.OpenI)OTU(FQIC_4302_11_Reset)OTL(S4352_Phase_Circulation.Adv);
   12: XIC(S4352_Phase_Circulation.StepBit.7)XIC(SV_S52_2.OpenI)[GRT(S4352_Phase_Circulation.RealParameters[0],0) OTL(S4352_Phase_Circulation.Adv) ,MUL(S4352_Phase_Circulation.RealParameters[0],60000,S52_Circulation_Timer.PRE) ];
   13: CPT(S52CirculationRemMins,(S52_Circulation_Timer.PRE-S52_Circulation_Timer.ACC)/60000);
   14: XIC(S4352_Phase_Circulation.StepBit.8)[OTL(S4352_Phase_Circulation.Adv) ,OTL(Circulation_Timer_Continue) ];
   15: XIC(Circulation_Timer_Continue)XIO(S52_Circulation_Timer.DN)TON(S52_Circulation_Timer,?,?);
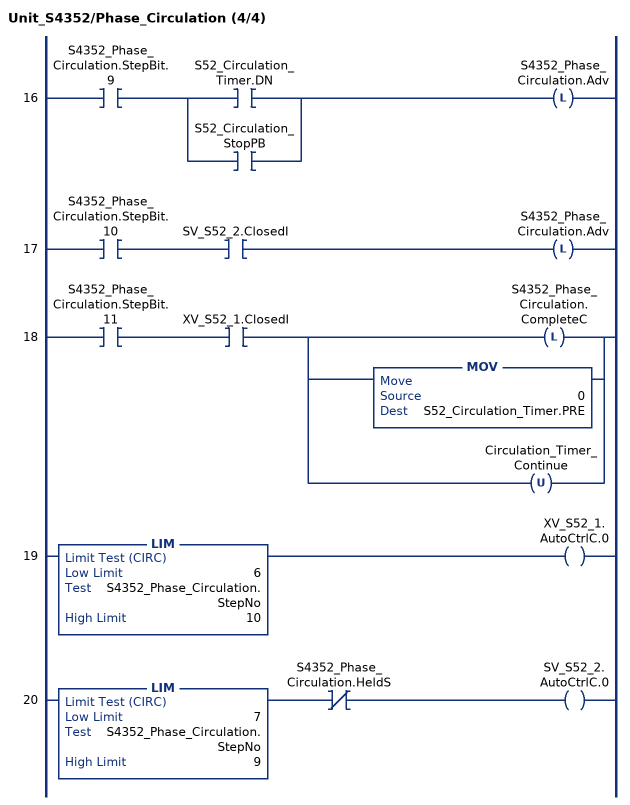
   16: XIC(S4352_Phase_Circulation.StepBit.9)[XIC(S52_Circulation_Timer.DN) ,XIC(S52_Circulation_StopPB) ]OTL(S4352_Phase_Circulation.Adv);
   17: XIC(S4352_Phase_Circulation.StepBit.10)XIC(SV_S52_2.ClosedI)OTL(S4352_Phase_Circulation.Adv);
   18: XIC(S4352_Phase_Circulation.StepBit.11)XIC(XV_S52_1.ClosedI)[OTL(S4352_Phase_Circulation.CompleteC) ,MOV(0,S52_Circulation_Timer.PRE) ,OTU(Circulation_Timer_Continue) ];
   19: LIM(6,S4352_Phase_Circulation.StepNo,10)OTE(XV_S52_1.AutoCtrlC.0);
   20: LIM(7,S4352_Phase_Circulation.StepNo,9)XIO(S4352_Phase_Circulation.HeldS)OTE(SV_S52_2.AutoCtrlC.0);
END_ROUTINE
